TYPE ST_HMI_BUTTON_IN :
STRUCT
	bClick	: BOOL;
END_STRUCT
END_TYPE

(* stored: Version 1.1.0.1
   DUT ST_HMI_BUTTON_IN: Id {6cca55ce-eaa1-4245-be3b-dee191b16f02} *)
